FUNCTION_BLOCK E_N_TABLE (* Generation of a finite train of sperate events *)
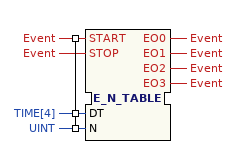
  EVENT_INPUT
    START WITH DT, N;
    STOP;
  END_EVENT
  EVENT_OUTPUT
    EO0;
    EO1;
    EO2;
    EO3;
  END_EVENT
  VAR_INPUT
    DT : ARRAY [0..3] OF TIME;
    N : UINT;
  END_VAR
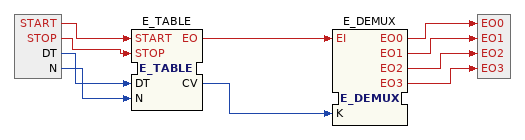
  FBS
    E_TABLE : iec61499::events::E_TABLE;
    E_DEMUX : iec61499::events::E_DEMUX;
  END_FBS
  EVENT_CONNECTIONS
    START TO E_TABLE.START;
    STOP TO E_TABLE.STOP;
    E_TABLE.EO TO E_DEMUX.EI;
    E_DEMUX.EO0 TO EO0;
    E_DEMUX.EO1 TO EO1;
    E_DEMUX.EO2 TO EO2;
    E_DEMUX.EO3 TO EO3;
  END_CONNECTIONS
  DATA_CONNECTIONS
    DT TO E_TABLE.DT;
    N TO E_TABLE.N;
    E_TABLE.CV TO E_DEMUX.K;
  END_CONNECTIONS
END_FUNCTION_BLOCK
